Yaskawa INFORM job: MOVE_INTO_TUNNEL.JBI

/JOB
//NAME MOVE_INTO_TUNNEL
///FOLDERNAME IMPORTANT_JOBS
//POS
///NPOS 2,2,0,0,0,0
///TOOL 0
///POSTYPE ROBOT
///RECTAN
///RCONF 0,0,1,0,0,0,0,0,0,0,0,0,0,0,0,0,0,0,0,0,0,0,0,0
C00000=1961.335,0.063,151.266,-0.1275,-76.2674,0.1269
C00001=1960.999,-0.993,151.006,-0.0021,-76.0002,0.0019
///RCONF 0,0,0,0,0,0,0,0,0,0,0,0,0,0,0,0,0,0,0,0,0,0,0,0
BC00000=0.000
BC00001=2689.532
//INST
///DATE 2024/06/04 20:51
///ATTR SC,RW,RJ
////FRAME ROBOT
///GROUP1 RB1,BS1
NOP
SFTOF
WAIT SOUT#(57)=ON
CALL JOB:R1-HOME
MOVJ C00000 BC00000 VJ=50.00
MOVJ C00001 BC00001 VJ=50.00
WAIT SOUT#(58)=ON
END
